// TIA Portal V16 export
// export: Created 2021-07-03T21:22:43.003899Z, ExportSetting WithDefaults, DisplayName Totally Integrated Automation Portal, DisplayVersion V16, DisplayName TIA Portal Version Control Interface, DisplayVersion V16, DisplayName TIA Portal Openness, DisplayVersion V16, DisplayName STEP 7 Professional, DisplayVersion V16, DisplayName STEP 7 Safety, DisplayVersion V16, DisplayName WinCC Professional, DisplayVersion V16
TYPE "118MK2_RecipeEdit"
// stored: IsFailsafeCompliant false
   STRUCT
      SPARE0 { ExternalAccessible := 'False'; ExternalVisible := 'False'; ExternalWritable := 'False'} : Byte;   // Spare
      ACTIVE_RECIPE_E { ExternalAccessible := 'False'; ExternalVisible := 'False'; ExternalWritable := 'False'} : Byte := BYTE#16#01;   // Scratch Pad : Active Recipe, (1 to 15)
      REC_EJEC_DELAY_TIME_E { ExternalAccessible := 'False'; ExternalVisible := 'False'; ExternalWritable := 'False'} : Byte;   // Scratchpad: Ejector delay time - Unsigned 8 bit integer value. Range 0 to 50ms
      REC_EJEC_ON_TIME_E { ExternalAccessible := 'False'; ExternalVisible := 'False'; ExternalWritable := 'False'} : Byte;   // Scratchpad: Ejector on time - Unsigned 8 bit integer value. Range 1 to 50ms
      REC_ALG_BLINT_TH_E { ExternalAccessible := 'False'; ExternalVisible := 'False'; ExternalWritable := 'False'} : Word;   // Scratchpad: Algorithm blue intensity threshold - Unsigned 16 bit integer value. Range 60 to 10000mV
      REC_ALG_BLRD_DOFF_E { ExternalAccessible := 'False'; ExternalVisible := 'False'; ExternalWritable := 'False'} : Word;   // Scratchpad: Algorithm blue-red discrimination offset - Unsigned 16 bit integer value. Range 0 to 10000
      REC_ALG_BLRD_DRAT_E { ExternalAccessible := 'False'; ExternalVisible := 'False'; ExternalWritable := 'False'} : Word;   // Scratchpad: Algorithm blue-red discrimination ratio - Unsigned 16 bit integer value. Range 1 to 1000 (is gradient of 0.01 to 10.00)
      REC_VIB_FEED_SP_E { ExternalAccessible := 'False'; ExternalVisible := 'False'; ExternalWritable := 'False'} : Byte;   // Scratchpad: Vibratory feeder set-point, Unsigned 8 bit integer value. Range 0 to 100%
      REC_AUTO_FEED_CNTRL_E { ExternalAccessible := 'False'; ExternalVisible := 'False'; ExternalWritable := 'False'} : Bool;   // Scratchpad: Automatic feeder control - OFF(0) – No closed loop control, ON(1) – Closed loop control
      REC_RESERVED1_E { ExternalAccessible := 'False'; ExternalVisible := 'False'; ExternalWritable := 'False'} : Bool;   // Scratchpad: Reserved - Spare
      REC_RESERVED2_E { ExternalAccessible := 'False'; ExternalVisible := 'False'; ExternalWritable := 'False'} : Bool;   // Scratchpad: Reserved - Spare
      REC_RESERVED3_E { ExternalAccessible := 'False'; ExternalVisible := 'False'; ExternalWritable := 'False'} : Bool;   // Scratchpad: Reserved - Spare
      REC_RESERVED4_E { ExternalAccessible := 'False'; ExternalVisible := 'False'; ExternalWritable := 'False'} : Bool;   // Scratchpad: Reserved - Spare
      REC_RESERVED5_E { ExternalAccessible := 'False'; ExternalVisible := 'False'; ExternalWritable := 'False'} : Bool;   // Scratchpad: Reserved - Spare
      REC_RESERVED6_E { ExternalAccessible := 'False'; ExternalVisible := 'False'; ExternalWritable := 'False'} : Bool;   // Scratchpad: Reserved - Spare
      REC_RESERVED7_E { ExternalAccessible := 'False'; ExternalVisible := 'False'; ExternalWritable := 'False'} : Bool;   // Scratchpad: Reserved - Spare
      REC_GATE_POSITION_E { ExternalAccessible := 'False'; ExternalVisible := 'False'; ExternalWritable := 'False'} : Byte;   // Scratchpad: Gate position - Range 0 to 5, ‘0’ - No auto gate control, ‘1’ – Move gate to position 1(-2 +1mm), ‘2’ – Move gate to position 2(-4+2mm), ‘3’ – Move gate to position 3(-8+4mm), ‘4’ – Move gate to position 4(-16+8mm), ‘5’ – Move gate to position 5(-32+16mm)
      SPARE1 { ExternalAccessible := 'False'; ExternalVisible := 'False'; ExternalWritable := 'False'} : Byte;   // Spare
      SPARE2 { ExternalAccessible := 'False'; ExternalVisible := 'False'; ExternalWritable := 'False'} : Word;   // Spare
   END_STRUCT;
END_TYPE
